RoboDK station: CuttingShapes.rdk

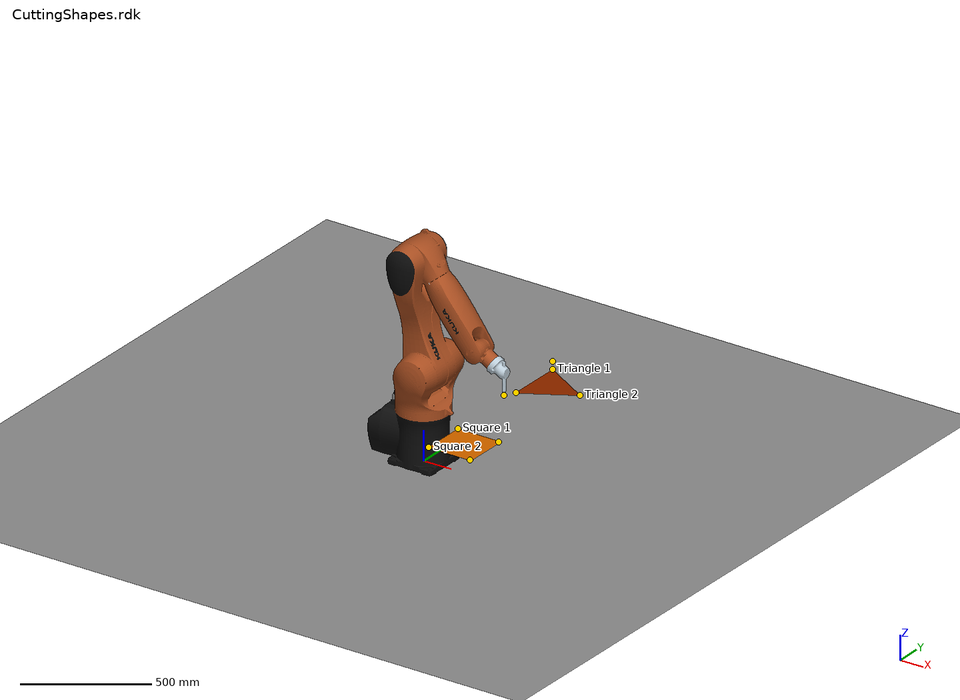
[picture v0: the station drawn from its stored meshes, robots at their saved joint values, targets as dots, program paths as lines]
Station CuttingShapes (saved by RoboDK 5.4.1). Poses are relative to the parent item; angles as X-Y-Z fixed-axis rotations.
Station parameters (name, value as stored): LIN64
  - frame KUKA KR 6 R900 sixx Base at (-207.87, 0, -62.35) mm
    - robot KUKA KR 6 R900 sixx: 6 axes, payload 6 kg, reach 901 mm, repeatability 0.03 mm, weight 52 kg
        modified DH rows (alpha deg, a mm, theta deg, d mm): 0, 0, 0, 400; -90, 25, 0, 0; 0, 455, -90, 0; -90, 35, 0, 420; 90, 0, 0, 0; -90, 0, 180, 80
        joint limits [-170, -190, -120, -185, -120, -350] to [170, 45, 156, 185, 120, 350]; home [0, -90, 90, 0, 0, 0]; saved at [-0.563, -97.056, 149.262, 178.71, 22.21, -179.087]
      - tool Pencil, TCP at (82.2, 0, 101.78) mm, rotated rx 0 ry 60 rz 0 deg, size 74.9 x 125 x 107.3 mm
    - object Triangle at (300, 300, 300) mm, rotated rx 0 ry 0 rz 180 deg, size 216.5 x 250 x 0 mm, geometry from Triangle.sld
    - object Square at (400, -300, 300) mm, size 200 x 200 x 0 mm, geometry from Square.sld
    - object Floor at (0, 0, 0) mm, size 3000 x 3000 x 0 mm, geometry from Floor.sld
    - target Triangle 1 (Cartesian target) at (300.47, 424.07, 300) mm, rotated rx 180 ry 0 rz 180 deg; joints [-66.529, -64.125, 124.381, 93.704, 52.753, -145.133] of KUKA KR 6 R900 sixx
    - target Triangle 2 (Cartesian target) at (514.41, 300.89, 300) mm, rotated rx 180 ry 0 rz 180 deg; joints [-37.084, -61.098, 118.784, 121.228, 37.639, -148.142] of KUKA KR 6 R900 sixx
    - target Triangle 3 (Cartesian target) at (301.4, 179.55, 300) mm, rotated rx 180 ry 0 rz 180 deg; joints [-44.133, -81.42, 153.14, 125.703, 47.954, -162.896] of KUKA KR 6 R900 sixx
    - target Square 1 (Cartesian target) at (301.73, -203.62, 300) mm, rotated rx 180 ry 0 rz 180 deg; joints [47.681, -79.801, 150.804, 58.752, -48.504, -18.745] of KUKA KR 6 R900 sixx
    - target Square 2 (Cartesian target) at (301.71, -397.51, 300) mm, rotated rx 180 ry 0 rz 180 deg; joints [64.998, -66.066, 127.913, 83.689, -52.154, -32.787] of KUKA KR 6 R900 sixx
    - target Square 3 (Cartesian target) at (494.3, -397.85, 300) mm, rotated rx 180 ry 0 rz 180 deg; joints [46.468, -56.904, 110.88, 73.301, -40.958, -40.577] of KUKA KR 6 R900 sixx
    - target Square 4 (Cartesian target) at (492.86, -205.55, 300) mm, rotated rx -180 ry 0 rz 180 deg; joints [28.631, -66.853, 129.33, 43.125, -37.375, -21.393] of KUKA KR 6 R900 sixx
    - target Retract_InspectA (Cartesian target) at (370.47, 2.5, 379.03) mm, rotated rx 180 ry 0 rz -180 deg; joints [-0.563, -97.056, 149.262, 178.71, 22.21, -179.087] of KUKA KR 6 R900 sixx
    - target App_InspectA (Cartesian target) at (595.41, 2.5, 584.69) mm, rotated rx 180 ry 0 rz -180 deg; joints [-0.299, -84.178, 103.493, 181.395, -10.689, -181.52] of KUKA KR 6 R900 sixx
  - Python program main (listed below)

--- Python program main ---
from robodk.robolink import *      # RoboDK's API
from robodk.robomath import *      # Math toolbox for robots
import cv2
import imutils

class ShapeDetector:
	def __init__(self):
		pass

	def detect(self, c):
		# initialize the shape name and approximate the contour
		shape = "unidentified"
		peri = cv2.arcLength(c, True)
		approx = cv2.approxPolyDP(c, 0.04 * peri, True)

		# if the shape is a triangle, it will have 3 vertices else it's a rectangle
		if len(approx) == 3:
			shape = "triangle"
		else:
			shape = "square"

		# return the name of the shape
		return shape

def getShape():
    webcam = cv2.VideoCapture(0)
    while True:
        _, frame = webcam.read()
        cv2.imshow('Webcam', frame)
        if cv2.waitKey(1) & 0xFF == ord('q'):
            break

    webcam.release()

    cv2.imshow('Webcam', frame)
    cv2.waitKey(0)

    cv2.destroyAllWindows()

    return frame

def detectShape():
    # load the image and resize it to a smaller factor so that
    # the shapes can be approximated better
    image = getShape()
    resized = imutils.resize(image, width=300)
    ratio = image.shape[0] / float(resized.shape[0])

    # convert the resized image to grayscale, blur it slightly,
    # and threshold it
    gray = cv2.cvtColor(resized, cv2.COLOR_BGR2GRAY)
    blurred = cv2.GaussianBlur(gray, (5, 5), 0)
    thresh = cv2.threshold(blurred, 60, 255, cv2.THRESH_BINARY)[1]

    # find contours in the thresholded image and initialize the
    # shape detector
    cnts = cv2.findContours(thresh.copy(), cv2.RETR_EXTERNAL, cv2.CHAIN_APPROX_SIMPLE)
    cnts = imutils.grab_contours(cnts)
    sd = ShapeDetector()

    # loop over the contours
    for c in cnts:
        # compute the center of the contour, then detect the name of the
        # shape using only the contour
        M = cv2.moments(c)
        cX = int((M["m10"] / M["m00"]) * ratio)
        cY = int((M["m01"] / M["m00"]) * ratio)
        shape = sd.detect(c)

        # multiply the contour (x, y)-coordinates by the resize ratio,
        # then draw the contours and the name of the shape on the image
        c = c.astype("float")
        c *= ratio
        c = c.astype("int")
        cv2.drawContours(image, [c], -1, (0, 255, 0), 2)
        cv2.putText(image, shape, (cX, cY), cv2.FONT_HERSHEY_SIMPLEX,
            0.5, (0, 0, 0), 2)

        # show the output image
        cv2.imshow("Image", image)
        cv2.waitKey(0)
    return shape

RL = Robolink()

robot = RL.Item('KUKA KR 6 R900 sixx')

app_InspectA = RL.Item('App_InspectA')
retract_InspectA = RL.Item('Retract_InspectA')

def moveRobot(shape):
    robot.MoveJ(app_InspectA)
    if shape == "triangle":
        moveTriangle()
    else:
        moveSquare()
    robot.MoveJ(retract_InspectA)

def moveTriangle():
    for i in range(1, 4):
        targetName = f"Triangle {i}"
        robot.MoveJ(RL.Item(targetName))
    robot.MoveJ(RL.Item("Triangle 1"))

def moveSquare():
    for i in range(1, 5):
        targetName = f"Square {i}"
        robot.MoveJ(RL.Item(targetName))
    robot.MoveJ(RL.Item("Square 1"))

for i in range(2):
    shape = detectShape()
    moveRobot(shape)
